(* IEC 61131-3 sources: ICSML/Codesys_V3/Functions, 12 files *)

(* ---- ARRBIN.pou ---- *)
(*#-#-#-#-#-#-#-#-#-#---Declaration---#-#-#-#-#-#-#-#-#-#-#-#-#*)

(*
	Helper function to write data from an array to a binary file. Can be used to write inference results or intermediate data.

	Parameters:
		filename: Absolute path to binary file. If file does not exist, it will be created. E.g: '/home/user/weights.bin'.
		bytes: Number of bytes to write. E.g for a 6x8 LREAL matrix: 6*8*SIZEOF(LREAL)
		src: Pointer to array from where the data should be read
		err (optional): Pointer to CmpErrors.RTS_IEC_RESULT to get errors
		overwrite (optional): Boolean on whether writing should be done in Overwrite or Append mode (default).

	Depends on CmpError and SysFile libraries.
*)
FUNCTION ARRBIN : DWORD
VAR_INPUT
	filename: STRING;
	bytes: DWORD;
	src: DWORD;
	err: POINTER TO CmpErrors.RTS_IEC_RESULT := 0;
	overwrite: BOOL := FALSE;
END_VAR
VAR
	file_handle: SysFile.RTS_IEC_HANDLE;
	bytes_written: DWORD;
END_VAR

(*#-#-#-#-#-#-#-#-#-#---Implementation---#-#-#-#-#-#-#-#-#-#-#-#-#*)

// Open file in write or append mode
IF overwrite = FALSE THEN
	file_handle := SysFileOpen(filename, SysFile.AM_APPEND_PLUS, err);
ELSE
	file_handle := SysFileOpen(filename, SysFile.AM_WRITE, err);
END_IF

// Read and copy bytes into array
bytes_written := SysFileWrite(file_handle, src, bytes, err);

// Close file
SysFileClose(file_handle);

(* ---- BINARR.pou ---- *)
(*#-#-#-#-#-#-#-#-#-#---Declaration---#-#-#-#-#-#-#-#-#-#-#-#-#*)

(*
	Helper function to load data from a binary file to an array. Can be used to load layer weights and biases.

	Parameters:
		filename: Absolute path to binary file. E.g: '/home/user/weights.bin'
		bytes: Number of bytes to read. E.g for a 6x8 LREAL matrix: 6*8*SIZEOF(LREAL)
		dst: Pointer to array where the data should be loaded
		err (optional): Pointer to CmpErrors.RTS_IEC_RESULT to get errors

	Depends on CmpError and SysFile libraries.
*)
FUNCTION BINARR : DWORD
VAR_INPUT
	filename: STRING;
	bytes: DWORD;
	dst: DWORD;
	err: POINTER TO CmpErrors.RTS_IEC_RESULT := 0;
END_VAR
VAR
	file_handle: SysFile.RTS_IEC_HANDLE;
	bytes_read: DWORD;
END_VAR

(*#-#-#-#-#-#-#-#-#-#---Implementation---#-#-#-#-#-#-#-#-#-#-#-#-#*)

// Open file as read only
file_handle := SysFileOpen(filename, SysFile.AM_READ, err);

// Read and copy bytes into array
bytes_read := SysFileRead(file_handle, dst, bytes, err);

// Close file
SysFileClose(file_handle);

(* ---- BSTEP.pou ---- *)
(*#-#-#-#-#-#-#-#-#-#---Declaration---#-#-#-#-#-#-#-#-#-#-#-#-#*)

(*
	Binary Step Activation Function.
*)
FUNCTION BSTEP : REAL
VAR_INPUT
	input: REAL;
END_VAR
(*#-#-#-#-#-#-#-#-#-#---Implementation---#-#-#-#-#-#-#-#-#-#-#-#-#*)

IF input >= 0 THEN
	BSTEP := 1;
ELSE
	BSTEP := 0;
END_IF

(* ---- DOT.pou ---- *)
(*#-#-#-#-#-#-#-#-#-#---Declaration---#-#-#-#-#-#-#-#-#-#-#-#-#*)

(*
	Dot Product calculation function
*)
FUNCTION DOT : REAL
VAR_INPUT
	vectorA: POINTER TO REAL;
	vectorB: POINTER TO REAL;
	length: DINT;
END_VAR
VAR
	result: REAL := 0;
	index: DINT;
END_VAR

(*#-#-#-#-#-#-#-#-#-#---Implementation---#-#-#-#-#-#-#-#-#-#-#-#-#*)

FOR index := 0 TO length-1 DO
	result := result + vectorA[index] * vectorB[index];
END_FOR

DOT := result;

(* ---- ELU.pou ---- *)
(*#-#-#-#-#-#-#-#-#-#---Declaration---#-#-#-#-#-#-#-#-#-#-#-#-#*)

(*
	Exponential Linear Unit (ELU).

	Parameters:
		alpha: ELU alpha parameter for defining scaling of the function when input < 0
*)
FUNCTION ELU : REAL
VAR_INPUT
	input: REAL;
	alpha: REAL := 1;
END_VAR

(*#-#-#-#-#-#-#-#-#-#---Implementation---#-#-#-#-#-#-#-#-#-#-#-#-#*)

IF input > 0 THEN
	ELU := input;
ELSE
	ELU := alpha * (EXP(input) - 1);
END_IF

(* ---- LIN.pou ---- *)
(*#-#-#-#-#-#-#-#-#-#---Declaration---#-#-#-#-#-#-#-#-#-#-#-#-#*)

(*
	Linear Activation Function with slope.
*)
FUNCTION LIN : REAL
VAR_INPUT
	input: REAL;
	slope: REAL := 1;
END_VAR
(*#-#-#-#-#-#-#-#-#-#---Implementation---#-#-#-#-#-#-#-#-#-#-#-#-#*)

LIN := slope * input;

(* ---- LRELU.pou ---- *)
(*#-#-#-#-#-#-#-#-#-#---Declaration---#-#-#-#-#-#-#-#-#-#-#-#-#*)

(*
	Leaky Rectified Linear Unit (ReLU) activation function.
*)
FUNCTION LRELU : REAL
VAR_INPUT
	input: REAL;
END_VAR

(*#-#-#-#-#-#-#-#-#-#---Implementation---#-#-#-#-#-#-#-#-#-#-#-#-#*)

IF input >= 0 THEN
	LRELU := input;
ELSE
	LRELU := 0.01 * input;
END_IF

(* ---- RELU.pou ---- *)
(*#-#-#-#-#-#-#-#-#-#---Declaration---#-#-#-#-#-#-#-#-#-#-#-#-#*)

(*
	Rectified Linear Unit (ReLU) activation function.

	Parameters:
		alpha: Slope to multiply input with if input is less than 0. Default is 0.
*)
FUNCTION RELU : REAL
VAR_INPUT
	input: REAL;
	alpha: REAL := 0;
END_VAR

(*#-#-#-#-#-#-#-#-#-#---Implementation---#-#-#-#-#-#-#-#-#-#-#-#-#*)

IF input >= 0 THEN
	RELU := input;
ELSE
	RELU := input * alpha;
END_IF

(* ---- SIG.pou ---- *)
(*#-#-#-#-#-#-#-#-#-#---Declaration---#-#-#-#-#-#-#-#-#-#-#-#-#*)

(*
Sigmoid Function
*)
FUNCTION SIG : REAL
VAR_INPUT
	input: REAL;
END_VAR
(*#-#-#-#-#-#-#-#-#-#---Implementation---#-#-#-#-#-#-#-#-#-#-#-#-#*)

SIG := 1 / (1+EXP(-input));

(* ---- SOFTMAX.pou ---- *)
(*#-#-#-#-#-#-#-#-#-#---Declaration---#-#-#-#-#-#-#-#-#-#-#-#-#*)

(*
	Softmax Activation Function.

	Parameters:
		input: Array of REAL to calculate the probability distribution on.
		output: Array of REAL to store results.
*)
FUNCTION SOFTMAX : INT
VAR_INPUT
	input: POINTER TO REAL;
	output: POINTER TO REAL;
	length: DINT;
END_VAR
VAR
	sum: REAL := 0;
	index: DINT;
END_VAR

(*#-#-#-#-#-#-#-#-#-#---Implementation---#-#-#-#-#-#-#-#-#-#-#-#-#*)

// Calculate sum of EXP(input[index])
FOR index := 0 TO length-1 DO
	sum := sum + EXP(input[index]);
END_FOR

// Calculate probabilities
FOR index := 0 TO length-1 DO
	output[index] := EXP(input[index]) / sum;
END_FOR

(* ---- SWISH.pou ---- *)
(*#-#-#-#-#-#-#-#-#-#---Declaration---#-#-#-#-#-#-#-#-#-#-#-#-#*)

(*
	Swish Activation Function.
*)
FUNCTION SWISH : REAL
VAR_INPUT
	input: REAL;
END_VAR
(*#-#-#-#-#-#-#-#-#-#---Implementation---#-#-#-#-#-#-#-#-#-#-#-#-#*)

//SWISH := input * SIG(input);
SWISH := input/(1-EXP(-input));

(* ---- TANH.pou ---- *)
(*#-#-#-#-#-#-#-#-#-#---Declaration---#-#-#-#-#-#-#-#-#-#-#-#-#*)

(*
	Tanh activation function.
*)
FUNCTION TANH : REAL
VAR_INPUT
	input: REAL;
END_VAR
(*#-#-#-#-#-#-#-#-#-#---Implementation---#-#-#-#-#-#-#-#-#-#-#-#-#*)

//TANH := 2 * SIG(2*input) - 1;
TANH := (2 / (1 + EXP(-2*input))) - 1;
